TYPE (* IEC61131-3, Table 14#5 *)
  (* Standard: 1131-3 *)
  (* Version 0.0, 10/1/2026, Schneider Electric, Template *)
  PACKAGE Main;
  {SET_ATTRIBUTE(nxtDataType, tRPzkA71YZLpXBQsWDVLI5szmWdUitrxpXrIevJ3l/0GXoM6PmDfR1CTPkQcXzAC)}
  dtArray : ARRAY [0..9] OF INT;
END_TYPE
